(*
Nazwa:			E_GripperScrewerState
Opis:			Stan zakecarki szczekowej
Wersja:			v0.1
Data:			2023-10-10
Autor:			TW
Urzadzenia:		
Konfiguracja:	
Info:
*)

TYPE E_CapPreScrewer :
(	
	eReady							:= 10,
	ePreparingToPick				:= 20,			
	ePicking						:= 30,
	eVacumCheckPart1				:= 40,
	eVacumCheckPart2				:= 50,
	eVacumCheckPart3				:= 50,
	eVacumCheckPart4				:= 60,
	eTransferingVertical			:= 70,
	eTransferingHorizontal			:= 80,
	eAxisGearIn						:= 82,
	eVerticalDownToCatchPos			:= 90,
	ePositionOverBottle				:= 95,	
	eCatching						:= 100,		
	ePlacing						:= 110,
	eStrawCatcherBack				:= 120,
	eFinding						:= 130,
	eFindingStop					:= 140,
	ePreScrewing					:= 145,
	eScrewing						:= 150,
	eScrewingStop					:= 160,
	eFinished						:= 170,
	eGearOut						:= 175,
	                        		
	eReturning1						:= 180,
	eReturning2						:= 190,
                            		
			                	
	eDone							:= 200,
	eNotDone						:= 300
	


	
):= eReady;
END_TYPE

(* stored: Version 1.2.0.0, ProductVersion 3.1.4026.13, FileIdentifier 838c305df3f398fe0580ecac3e166930ac12758d, FileSignature 3368d61a33ff26aeaf57ecdd8d62d5e0123b9901f3df66cda4b4a294455fe8dc2e55488430102846c6bc908e093618da081af87e6a02b40904f2a284c6e6c948b3c1ec32d5c05d35602fed0083e0503ac1dd53cc35c80b44a9d1a0fb3e048da3e28a6f19d36149c2280acbb6664b788d2ed82896314f06022773c314f3a7966956b6d6bd6ce95dcb083a0c8ca0169cc930f9f5c70b49d2d88b2bfd614ee402261a61ecc10975e930d7c1b0a5f1ca2a82b11e248d333bc57889630b2f52f7c1abb2dfdb901922435c99ca4bdd94d252d979907a4d712f589061a3daf4238779e1f4e789f576c964038e8df512b0c39d7357a5d817292e8034b66863ac3ff30aaa
   DUT E_CapPreScrewer: Id {c2c880b5-b2d6-44a6-b076-b3c6c7bc5cd7} *)
